TYPE ST_HE_SolidAttenuatorHolderSettings :
STRUCT
    bEnabled : BOOL;
    fbBeamYInHolderCoordinates : FB_QuantityLREALPublic(Units := 'mm');
END_STRUCT
END_TYPE

(* stored: Version 1.1.0.1
   DUT ST_HE_SolidAttenuatorHolderSettings: Id {6d821e5e-5add-4e13-9ca9-0e3a732a33d1} *)
